(* PLC project Unnamed, Unknown Unnamed 1 *)
(* stored: creationDateTime 2023-03-19T23:09:43, modificationDateTime 2023-03-22T04:27:15 *)

PROGRAM Industrial_Automation_practice_Saw_Fan_Oil_pump
  VAR_IN_OUT
    Saw : BOOL;  (* turns on when start_button is pressed *)
  END_VAR
  VAR_OUTPUT
    Fan : BOOL;  (* turns on when start_button is pressed *)
    Oil_Pump : BOOL;  (* turns on when start_button is pressed *)
  END_VAR
  VAR_INPUT
    Start_Button : BOOL := 1;  (* turns on the saw, fan, and oiil_pump *)
  END_VAR
  VAR
    SR0 : SR;
    Saw_run_20s : BOOL;  (* latches when saw has been on for 20s *)
    SR1 : SR;
  END_VAR
  VAR_INPUT
    saw_off : BOOL := 0;  (* turns off Saw *)
  END_VAR
  VAR
    SR2 : SR;
  END_VAR
  VAR_INPUT
    Fan_reset_button : BOOL := 0;  (* only allow for fan reset when saw has been on for more than 20s and saw is off *)
    Saw_run_20s_reset : BOOL := 0;  (* resets Saw_run_20s_latch *)
  END_VAR
  VAR
    R_TRIG0 : R_TRIG;
    TON0 : TON;
    TON1 : TON;
    TON2 : TON;
    SR3 : SR;
  END_VAR
  VAR  (* added by the conversion: wires and edge detectors of the diagram *)
    _NOT19_OUT : BOOL;
    _AND6_OUT : BOOL;
    _AND23_OUT : BOOL;
  END_VAR

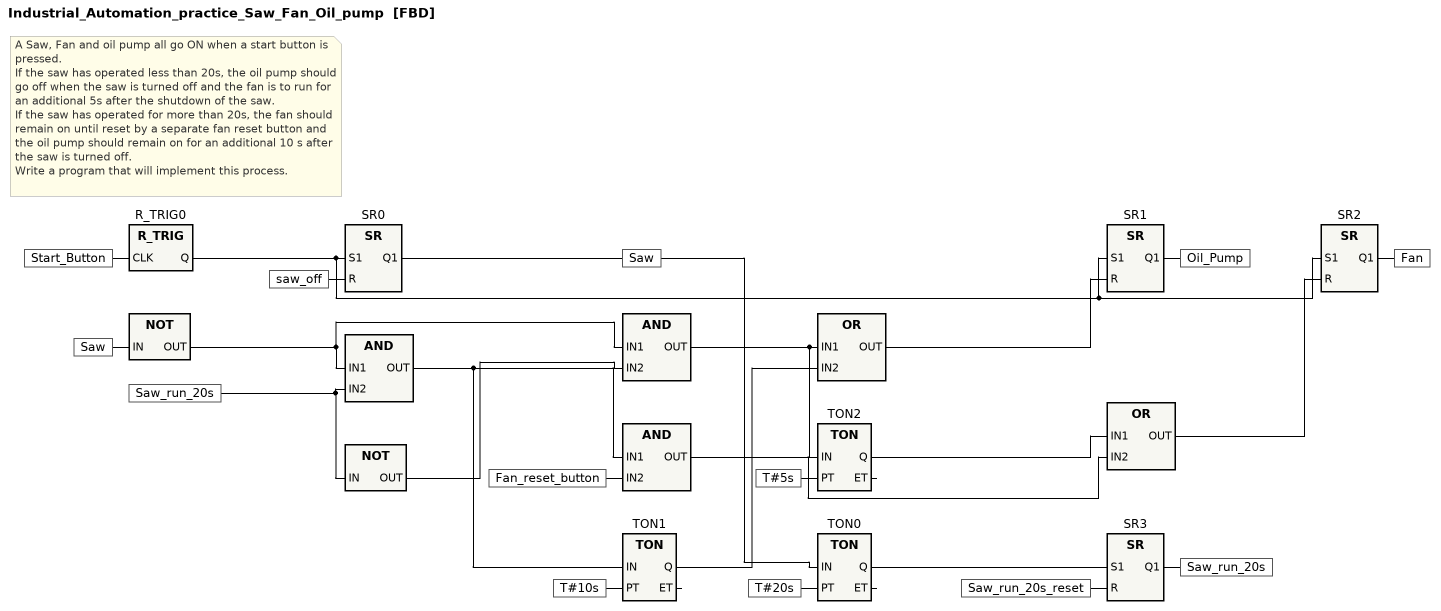
(* FBD diagram, written out as Structured Text *)
(* A Saw, Fan and oil pump all go ON when a start button is pressed.
    If the saw has operated less than 20s, the oil pump should go off when the saw is turned off and the fan is to run for an additional 5s after the shutdown of the saw.
    If the saw has operated for more than 20s, the fan should remain on until reset by a separate fan reset button and the oil pump should remain on for an additional 10 s after the saw is turned off.
    Write a program that will implement this process. *)
R_TRIG0(CLK := Start_Button);
SR0(S1 := R_TRIG0.Q, R := saw_off);
Saw := SR0.Q1;
TON0(IN := Saw, PT := T#20s);
SR3(S1 := TON0.Q, R := Saw_run_20s_reset);
Saw_run_20s := SR3.Q1;
_NOT19_OUT := NOT Saw;
_AND6_OUT := _NOT19_OUT AND NOT Saw_run_20s;
_AND23_OUT := _NOT19_OUT AND Saw_run_20s;
TON1(IN := _AND23_OUT, PT := T#10s);
SR1(S1 := R_TRIG0.Q, R := _AND6_OUT OR TON1.Q);
Oil_Pump := SR1.Q1;
TON2(IN := _AND6_OUT, PT := T#5s);
SR2(S1 := R_TRIG0.Q, R := TON2.Q OR _AND23_OUT AND Fan_reset_button);
Fan := SR2.Q1;
END_PROGRAM

CONFIGURATION Config0
  RESOURCE Res0 ON PLC
    TASK task0(INTERVAL := T#20ms, PRIORITY := 0);
    PROGRAM instance0 WITH task0 : Industrial_Automation_practice_Saw_Fan_Oil_pump;
  END_RESOURCE
END_CONFIGURATION
